(* IEC 61131-3 sources: ICSML/Codesys_V3/Function Blocks/Swish_L.pou, 1 file *)

(* ---- Swish_L.pou ---- *)
(*#-#-#-#-#-#-#-#-#-#---Declaration---#-#-#-#-#-#-#-#-#-#-#-#-#*)

(*
	Swish Activation Layer
*)
FUNCTION_BLOCK PUBLIC Swish_L IMPLEMENTS Activation
VAR
	// Input and Output dataMem variables
	input_i: dataMem;
	output_i: dataMem;
END_VAR
(*#-#-#-#-#-#-#-#-#-#---Implementation---#-#-#-#-#-#-#-#-#-#-#-#-#*)
